// Mitsubishi GX Works2 project: HMI PLC 연습문제 코드   PLC: Q03UDV

PROGRAM MAIN
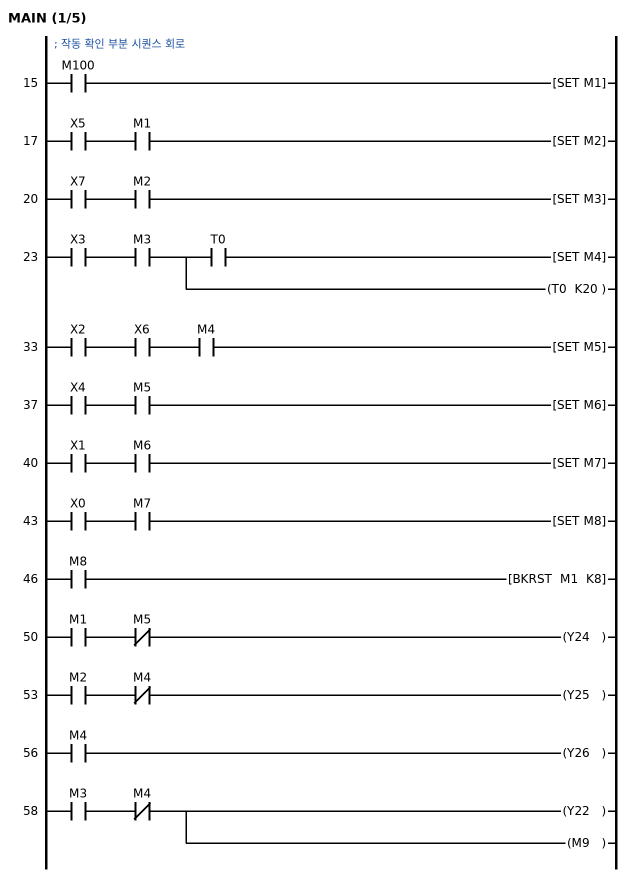
; 작동 확인 부분 시퀀스 회로
15    LD      M100
      SET     M1
17    LD      X5
      AND     M1
      SET     M2
20    LD      X7
      AND     M2
      SET     M3
23    LD      X3
      AND     M3
      MPS
      AND     T0
      SET     M4
      MPP
      OUT     T0 K20
33    LD      X2
      AND     X6
      AND     M4
      SET     M5
37    LD      X4
      AND     M5
      SET     M6
40    LD      X1
      AND     M6
      SET     M7
43    LD      X0
      AND     M7
      SET     M8
46    LD      M8
      BKRST   M1 K8
50    LD      M1
      ANI     M5
      OUT     Y24
53    LD      M2
      ANI     M4
      OUT     Y25
56    LD      M4
      OUT     Y26
58    LD      M3
      ANI     M4
      OUT     Y22
      OUT     M9
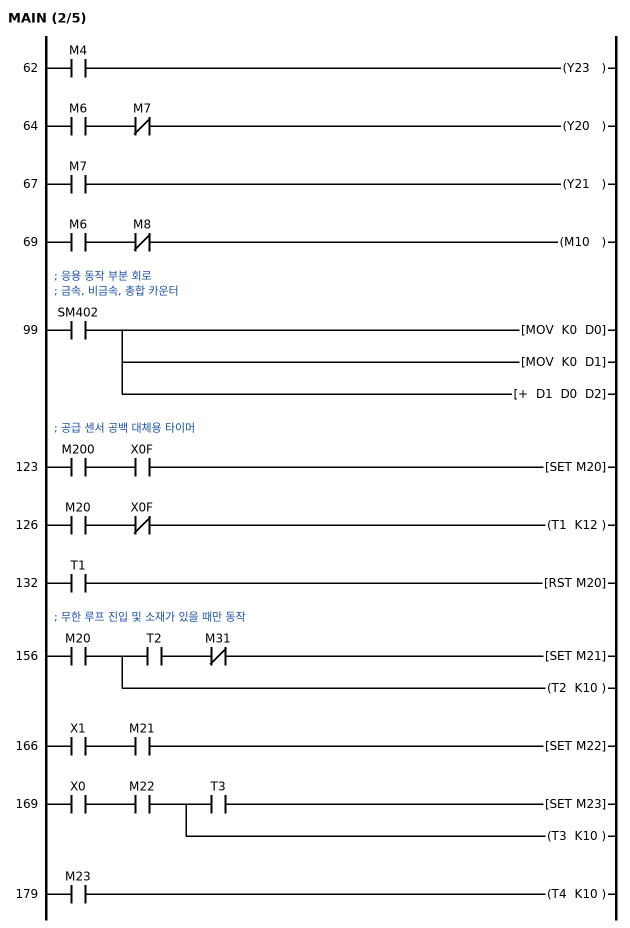
62    LD      M4
      OUT     Y23
64    LD      M6
      ANI     M7
      OUT     Y20
67    LD      M7
      OUT     Y21
69    LD      M6
      ANI     M8
      OUT     M10
; 응용 동작 부분 회로
; 금속, 비금속, 총합 카운터
99    LD      SM402
      MOV     K0 D0
      MOV     K0 D1
      +       D1 D0 D2
; 공급 센서 공백 대체용 타이머
123   LD      M200
      AND     X0F
      SET     M20
126   LD      M20
      ANI     X0F
      OUT     T1 K12
132   LD      T1
      RST     M20
; 무한 루프 진입 및 소재가 있을 때만 동작
156   LD      M20
      MPS
      AND     T2
      ANI     M31
      SET     M21
      MPP
      OUT     T2 K10
166   LD      X1
      AND     M21
      SET     M22
169   LD      X0
      AND     M22
      MPS
      AND     T3
      SET     M23
      MPP
      OUT     T3 K10
179   LD      M23
      OUT     T4 K10
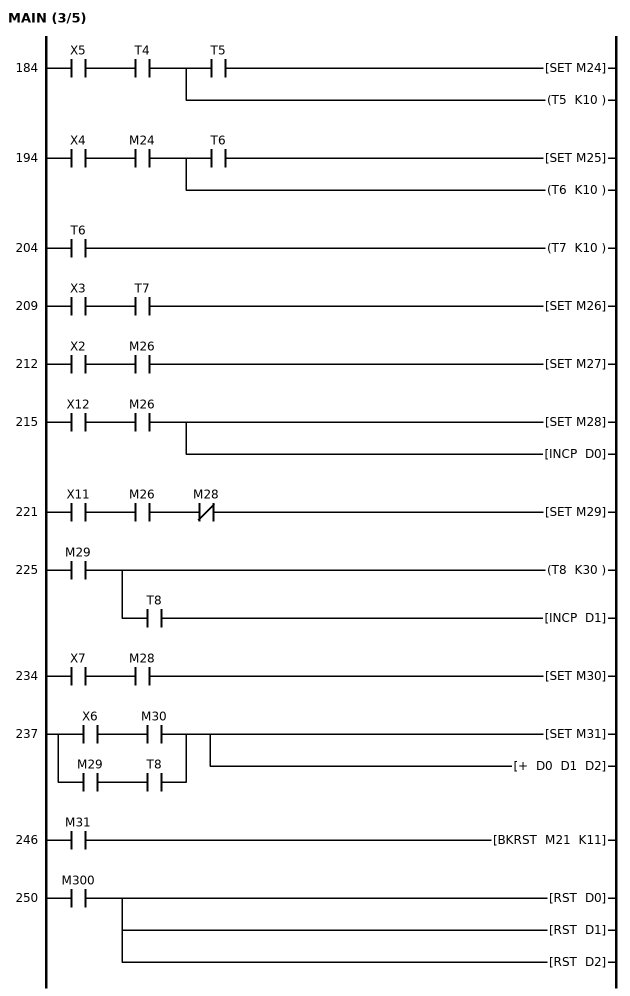
184   LD      X5
      AND     T4
      MPS
      AND     T5
      SET     M24
      MPP
      OUT     T5 K10
194   LD      X4
      AND     M24
      MPS
      AND     T6
      SET     M25
      MPP
      OUT     T6 K10
204   LD      T6
      OUT     T7 K10
209   LD      X3
      AND     T7
      SET     M26
212   LD      X2
      AND     M26
      SET     M27
215   LD      X12
      AND     M26
      SET     M28
      INCP    D0
221   LD      X11
      AND     M26
      ANI     M28
      SET     M29
225   LD      M29
      OUT     T8 K30
      AND     T8
      INCP    D1
234   LD      X7
      AND     M28
      SET     M30
237   LD      X6
      AND     M30
      LD      M29
      AND     T8
      ORB
      SET     M31
      +       D0 D1 D2
246   LD      M31
      BKRST   M21 K11
250   LD      M300
      RST     D0
      RST     D1
      RST     D2
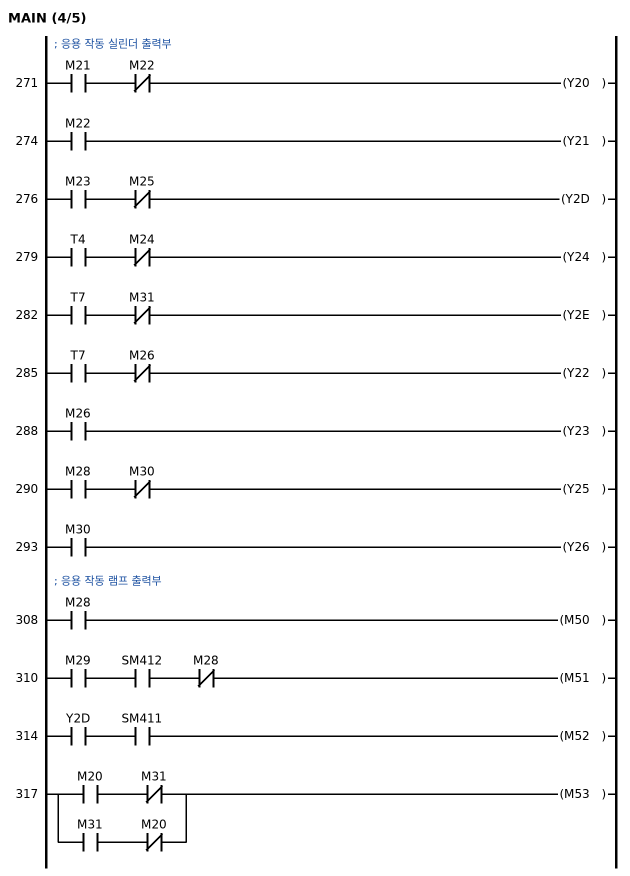
; 응용 작동 실린더 출력부
271   LD      M21
      ANI     M22
      OUT     Y20
274   LD      M22
      OUT     Y21
276   LD      M23
      ANI     M25
      OUT     Y2D
279   LD      T4
      ANI     M24
      OUT     Y24
282   LD      T7
      ANI     M31
      OUT     Y2E
285   LD      T7
      ANI     M26
      OUT     Y22
288   LD      M26
      OUT     Y23
290   LD      M28
      ANI     M30
      OUT     Y25
293   LD      M30
      OUT     Y26
; 응용 작동 램프 출력부
308   LD      M28
      OUT     M50
310   LD      M29
      AND     SM412
      ANI     M28
      OUT     M51
314   LD      Y2D
      AND     SM411
      OUT     M52
317   LD      M20
      ANI     M31
      LD      M31
      ANI     M20
      ORB
      OUT     M53
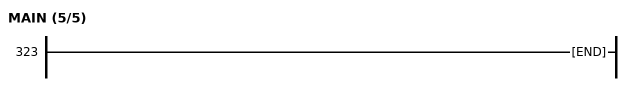
323   END
END_PROGRAM
